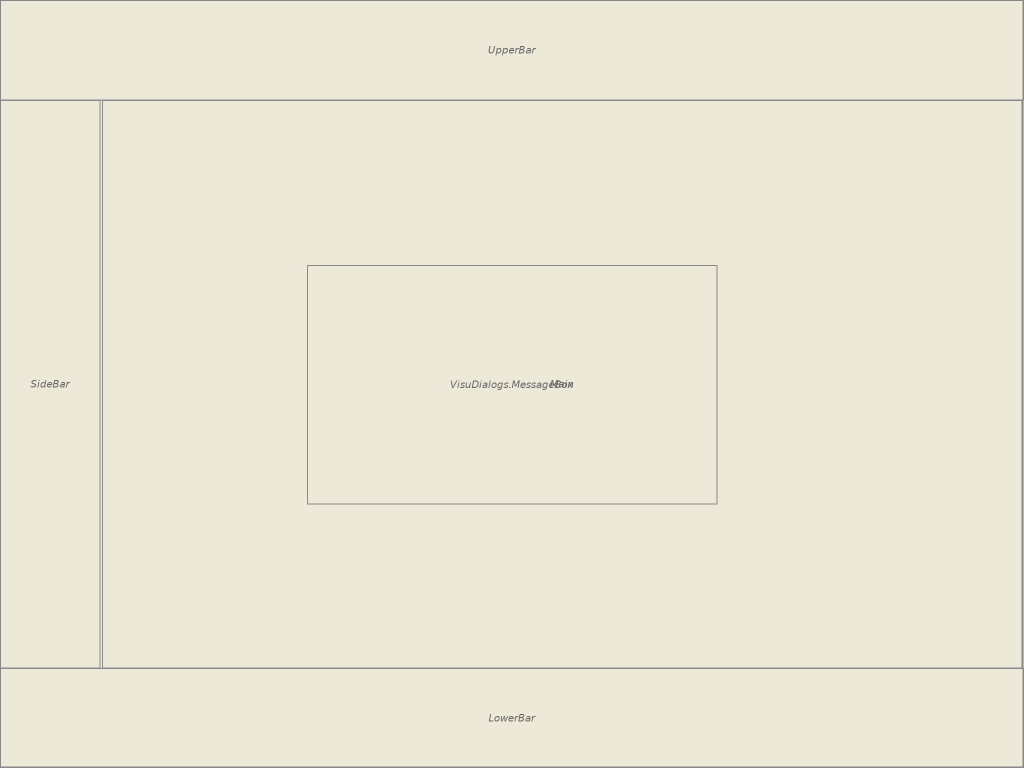
VISUALIZATION BasePage  // 1024x768
    Frame (0,0 1024x100)
        shows UpperBar()
    Frame (0,668 1024x100)
        shows LowerBar()
    Frame (0,100 100x568)
        shows SideBar()
    Frame (102,100 920x568), frame switch variable: GVL_HMI.iMainFrame
        shows Main()
        shows Manual()
        shows Setting()
        shows Model()
        shows Data()
        shows Alarm()
    Frame (307,265 410x239), invisible if: not bCallMessageBox
        shows VisuDialogs.MessageBox(eType := VisuDialogs.MessageBoxDialog_Types.OK_CANCEL, sTitle := sCurrentTitle, sMessageTxt := sCurrentMessage)
        OnMouseClick: execute { bCallMessageBox := false; }
END_VISUALIZATION

(* stored: Version 1.1.0.1
   Visu BasePage: Id {c9260f84-caf9-475b-97e2-b067f5654d28} *)
